ADAPTER AR (* unidirectional Adapter Interface for 1 Event and 1 Real *)
  (* Standard: 61499-1; Description: Copyright (c) 2026 HR Agrartechnik GmbH This program and the accompanying materials are made available under the terms of the Eclipse Public License 2.0 which is available at https://www.eclipse.org/legal/epl-2.0/ SPDX-License-Identifier: EPL-2.0 *)
  (* Version 1.0, 2026-01-17, Franz Höpfinger, HR Agrartechnik GmbH, Initial Version *)
  PACKAGE adapter::types::unidirectional;
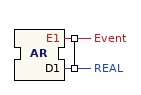
  EVENT_OUTPUT
    E1 WITH D1; (* Indication (or Request) *)
  END_EVENT
  VAR_OUTPUT
    D1 : REAL; (* Indication (or Request) Data from Plug *)
  END_VAR
END_ADAPTER
